FUNCTION Convert_SINT_TO_UDINT : Hresult
VAR_INPUT
	in : SINT;
	out : REFERENCE TO UDINT;
END_VAR
VAR
	converted : UDINT;
END_VAR
VAR CONSTANT
	INCOMPATIBLE : HRESULT := 16#9811070E;
END_VAR

converted := SINT_TO_UDINT(in);

IF (UDINT_TO_SINT(converted) <> in) THEN
	Convert_SINT_TO_UDINT := INCOMPATIBLE;
	RETURN;
END_IF

out := converted;

END_FUNCTION

(* stored: Version 1.1.0.1, ProductVersion 3.1.4024.12
   POU Convert_SINT_TO_UDINT: Id {15711023-6716-43fc-837d-338862350acb}, SpecialFunc None *)
